{attribute addProperty BoxType "EM7004-0000-0017"}
{attribute addProperty Id "StatusAT %I*Status_CBD542B4162"}
{attribute addProperty CRC "1539971487"}
{attribute addProperty SizeInBites "16"}
{attribute addProperty SizeInBytes "2"}
TYPE PLS_Inputs_5BCA199F :
STRUCT
	{attribute addProperty Name "Status"}
	Status AT %I* : Status_CBD542B4;
END_STRUCT
END_TYPE

(* stored: Version 1.2.0.0, ProductVersion 3.1.4024.9
   DUT PLS_Inputs_5BCA199F: Id {851c8542-eea7-4d4a-b642-c983d8a726c7} *)
